# EPICS substitutions: modules/event/evrSupport/Db/ioc/IOC-IN20-LS16evr.substitutions
#==============================================================================
#
# Abs:  LCLS EVR IOC records for IN20 LS16
#
# Name: IOC-IN20-LS16evr.substitutions
#
#==============================================================================
#
file evrLSXX.db
{
pattern { DEVICE        }
	{ EVR:IN20:LS16 }
}
